FUNCTION_BLOCK Motor
VAR_INPUT
END_VAR
VAR_OUTPUT
END_VAR
VAR
END_VAR

END_FUNCTION_BLOCK

(* stored: Version 1.1.0.1
   POU Motor: Id {ed772034-5018-4374-95a7-2d8f3f029229}, SpecialFunc None *)
